FUNCTION_BLOCK PUBLIC FB_Pizza
VAR_INPUT
END_VAR
VAR_OUTPUT
END_VAR
VAR
	eStyle		: E_PizzaStyle;
	bBroccoli	: BOOL;
	bCheese		: BOOL;
	bSalami		: BOOL;
END_VAR

PROPERTY PUBLIC bHasBroccoli : BOOL
GET
bHasBroccoli := this^.bBroccoli;
END_GET
SET
this^.bBroccoli := bHasBroccoli;
END_SET
END_PROPERTY

PROPERTY PUBLIC bHasCheese : BOOL
GET
bHasCheese := this^.bCheese;
END_GET
SET
this^.bCheese := bHasCheese;
END_SET
END_PROPERTY

PROPERTY PUBLIC bHasSalami : BOOL
GET
bHasSalami := this^.bSalami;
END_GET
SET
this^.bSalami := bHasSalami;
END_SET
END_PROPERTY

PROPERTY PUBLIC ePizzaStyle : E_PizzaStyle
GET
ePizzaStyle := this^.eStyle;
END_GET
SET
this^.eStyle := ePizzaStyle;
END_SET
END_PROPERTY

METHOD FB_init : BOOL
VAR_INPUT
	bInitRetains	: BOOL; // if TRUE, the retain variables are initialized (warm start / cold start)
	bInCopyCode		: BOOL;  // if TRUE, the instance afterwards gets moved into the copy code (online change)
	ePizzaStyle		: E_PizzaStyle;
	bHasBroccoli	: BOOL;
	bHasCheese 		: BOOL;
	bHasSalami		: BOOL;
END_VAR
THIS^.eStyle := ePizzaStyle;
THIS^.bBroccoli := bHasBroccoli;
THIS^.bCheese := bHasCheese;
this^.bSalami := bHasSalami;
END_METHOD

METHOD PUBLIC GetPrice : LREAL
IF (THIS^.eStyle = E_PizzaStyle.eItalian) THEN
	GetPrice := 4.5;
ELSIF (THIS^.eStyle = E_PizzaStyle.eAmerican) THEN
	GetPrice := 4.2;
ELSE
	GetPrice := 0;
	RETURN;
END_IF
IF (THIS^.bBroccoli) THEN
	GetPrice := GetPrice + 0.8;
END_IF
IF (THIS^.bCheese) THEN
	GetPrice := GetPrice + 1.1;
END_IF
IF (THIS^.bSalami) THEN
	GetPrice := GetPrice + 1.4;
END_IF
END_METHOD

END_FUNCTION_BLOCK

(* stored: Version 1.1.0.1, ProductVersion 3.1.4022.12
   POU FB_Pizza: Id {4112eb09-a32b-497d-9a14-4ebf43d24a50}, SpecialFunc None
   Property bHasBroccoli: Id {d32b6276-dfdd-4987-9330-43d3a510e0cf}
   Get Get: Id {63a8cf99-0577-4f60-b5a3-2fe96a5797eb}
   Set Set: Id {8c899d30-a660-437f-959e-9d83415ecc7a}
   Property bHasCheese: Id {8418113b-d6cf-43fd-8adb-49b754bf0b3a}
   Get Get: Id {8d0a2ad2-f621-45bb-ac8c-79038cb60a80}
   Set Set: Id {c3b1c124-02e9-4c87-a2ea-583313aba593}
   Property bHasSalami: Id {2282c824-2d39-49b6-8802-0140441c439e}
   Get Get: Id {d713f99c-01ae-4946-addb-d518b6a927d1}
   Set Set: Id {4ce4d4b9-365d-49bc-bd4d-dabd52f340c3}
   Property ePizzaStyle: Id {e9ab37f1-76a3-42d0-b784-3e1d03c363de}
   Get Get: Id {96100350-a6d8-4995-93b4-19fcf65e6570}
   Set Set: Id {2e623bd7-11ff-40d4-ae50-6dcc0c160a07}
   Method FB_init: Id {1b070e03-28f9-4434-9eef-c36c4d33f58c}
   Method GetPrice: Id {03d31fdd-6e7c-41d0-95b7-2f6838ec1645} *)
